KUKA KRL data list: TPallet.dat

&ACCESS RVO1
&REL 5
&PARAM EDITMASK = *
DEFDAT  TPallet

ENDDAT
